(* CODESYS project SPT_Vision.library
   Company: Beckhoff Automation LLC
   DefaultNamespace: SPT_Vision
   Version: 3.0.0
   Placeholder: SPT Vision
   Title: SPT Vision

Project tree, tasks and I/O mapping:
  libraries: SPT Base Types, * (Beckhoff Automation LLC); Tc2_Standard, * (Beckhoff Automation GmbH); Tc2_System, * (Beckhoff Automation GmbH); Tc3_Module, * (Beckhoff Automation GmbH); Tc3_Vision, * (Beckhoff Automation GmbH); SPT Event Logger, * (Beckhoff Automation LLC); Tc3_EventLogger, * (Beckhoff Automation GmbH); Tc2_Utilities, * (Beckhoff Automation GmbH); Tc2_EtherCAT, * (Beckhoff Automation GmbH)
  DUTs/
  GVLs/
  POUs/
    program MAIN [ST]
  Project Information/
    function F_GetCompany [ST]
    function F_GetTitle [ST]
    function F_GetVersion [ST]
  Version/
    global variables Global_Version
  Vision/
    DUTs/
      data type E_VisionTools
      data type ST_BlobResults
      data type ST_CameraReadWrite
      data type ST_Image2Video
      data type ST_VisionResults
    GVLs/
      global variables GVL_CameraDefinitions
      global variables GVL_Image2Video
      global variables GVL_VisionColor
    HMI/
      data type ST_VisionBase_Command
      data type ST_VisionBase_Config
      data type ST_VisionBase_HMI
      data type ST_VisionBase_Status
    PLC Task/
      function block FB_PlcCameraBase [ST]: CreateEvents, CyclicLogic, GetResults, Reset, RunVision, TriggerImage
    VisionTask/
      function block FB_CameraParameterBuffer [ST]: AddData, BufferCount, GetData, ReadData, ResetData
      function block FB_VideoPlaybackControl [ST]: Busy, Error, ErrorID, CyclicLogic, InitComplete, Execute, OnAlarmRaised, SubscribedEvents, SubscribeEvents, UnsubscribeEvents, AddImage, AlarmDelayTime, CameraID, FramesPerSecond, ImageReductionFactor, ImageSourceDirectory, VideoOutputDirectory, WriteImage
      function block FB_VisionCameraBase [ST]: LightBackground, ExposureAddress, GainAddress, CyclicLogic, HMICommunication, ProcessImage, ReadParamUDINT, SetParamUDINT
      function block FB_VisionCameraDetection [ST]: ProcessImage, Initialize
      function block FB_VisionCameraMonitor [ST]: CameraID, FramesPerSecond, ImageSourceDirectory, VideoOutputDirectory, CyclicLogic, Initialize, ProcessImage
      interface I_CameraBase: CyclicLogic, ProcessImage
    global variables Parameters_Vision
  VISUs/
*)

// Vision/DUTs/E_VisionTools
{attribute 'qualified_only'}
{attribute 'strict'}
TYPE E_VisionTools :
(
	Blob,
	Contour,
	Color
);
END_TYPE

// Vision/DUTs/ST_BlobResults
TYPE ST_BlobResults :
	STRUCT
		Area		   : LREAL;
		CenterOfMass   : TcVnPoint2_LREAL;
		Circularity	   : LREAL;
		Convexity	   : LREAL;
		Eccentricity   : LREAL;
		ExtremePoint   : TcVnPoint2_LREAL;
		InertiaRatio   : LREAL;
		Moments		   : TcVnMoments;
		Orientation	   : TcVnRotatedRectangle;
		OrientationExp : TcVnRotatedRectangle;
		Perimeter	   : LREAL;
		Roundness	   : LREAL;
	END_STRUCT
END_TYPE

// Vision/DUTs/ST_CameraReadWrite
TYPE ST_CameraReadWrite :
	(*CameraCommand consists of Camera parameter address in HEX(byte)
	AND the data TO be written TO that address in decimal (UDINT).*)
	STRUCT
		CamAddress : UDINT;
		CamData	   : UDINT;
		Valid	   : BOOL;
	END_STRUCT
END_TYPE

// Vision/DUTs/ST_Image2Video
TYPE ST_Image2Video :
	STRUCT
		VideoPathSource : STRING;
		ImagePathSource : STRING;
		VideoFilename	: STRING;
		VideoCreate		: BOOL;
		VideoCreated	: BOOL;
		VideoFPS		: UINT;
		Heartbeat		: BOOL;
	END_STRUCT
END_TYPE

// Vision/DUTs/ST_VisionResults
{attribute 'pack_mode' := '1'}
TYPE ST_VisionResults :
	STRUCT
		x		 : LREAL; //x offset in image
		y		 : LREAL; //y offset in image
		c		 : LREAL; //Rotation about Z
		Pass	 : BOOL;  //Pass/Fail bit
		Distance : LREAL; //Distance in measurement
	END_STRUCT
END_TYPE

// Vision/HMI/ST_VisionBase_Command
TYPE ST_VisionBase_Command :
	STRUCT
		StartAquisition : BOOL;
		StopAquisition	: BOOL;
		Trigger			: BOOL;
	END_STRUCT
END_TYPE

// Vision/HMI/ST_VisionBase_Config
TYPE ST_VisionBase_Config :
	STRUCT
		Gain			  : UDINT;
		SetGain			  : BOOL;
		ReadGain		  : BOOL;
		ReadGainValue	  : UDINT;
		Exposure		  : UDINT;
		SetExposure		  : BOOL;
		ReadExposure	  : BOOL;
		ReadExposureValue : UDINT;
	END_STRUCT
END_TYPE

// Vision/HMI/ST_VisionBase_HMI
TYPE ST_VisionBase_HMI :
	STRUCT
		Config	: ST_VisionBase_Config;
		Command : ST_VisionBase_Command;
		Status	: ST_VisionBase_Status;
	END_STRUCT
END_TYPE

// Vision/HMI/ST_VisionBase_Status
 
TYPE ST_VisionBase_Status :
	STRUCT
		VisionRunning : BOOL;
		CameraState	  : ETcVnCameraState;
		ElementsFound : UDINT;
	END_STRUCT
END_TYPE

// Version/Global_Version
{attribute 'TcGenerated'}
{attribute 'no-analysis'}
{attribute 'linkalways'}
// This function has been automatically generated from the project information.
VAR_GLOBAL CONSTANT
	{attribute 'const_non_replaced'}
	stLibVersion_SPT_Vision : ST_LibVersion := (iMajor := 3, iMinor := 0, iBuild := 0, iRevision := 0, nFlags := 0, sVersion := '3.0.0');
END_VAR

// Vision/GVLs/GVL_CameraDefinitions
{attribute 'qualified_only'}
VAR_GLOBAL CONSTANT
	
	// Baseler ACE camera 
	// Analog Controls - Gain
	M180_GAIN_ADDRESS	   : UDINT := 16#00020024; // only writeable if Gain Auto is off (220-850)

	// Acquisition - Trigger
	M180_TRIGGER_MODE_ADDRESS	: UDINT := 16#00040204; // 0= Off 1 = On
	M180_TRIGGER_SOURCE_ADDRESS : UDINT := 16#00040244; // 0 = software 1 = line(hardware)

	// Acquisition - Exposure
	M180_EXPOSURE_TIME_ADDRESS : UDINT := 16#00040464; // 24-1000000us 

	// AOI Controls
	M180_WIDTH_ADDRESS	  : UDINT := 16#00030204; // 1 - Camera width based on Binning
	M180_HEIGHT_ADDRESS	  : UDINT := 16#00030224; // 1 - Camera height based on Binning
	M180_X_OFFSET_ADDRESS : UDINT := 16#00030244; // pixel offset to be used if the width is smaller than max-adjust view
	M180_Y_OFFSET_ADDRESS : UDINT := 16#00030264; // pixel offset to be used if the height is smaller than max-adjust view
END_VAR

// Vision/GVLs/GVL_Image2Video
{attribute 'qualified_only'}
VAR_GLOBAL
	NumberOfCameras	   : UINT := Parameters_Vision.MAX_NUMBER_CAMERAS;
	CameraData		   : ARRAY[1..Parameters_Vision.MAX_NUMBER_CAMERAS] OF ST_Image2Video;
END_VAR

// Vision/GVLs/GVL_VisionColor
{attribute 'qualified_only'}
{attribute 'strict'}
VAR_GLOBAL
	ColorWhite	 : TcVnVector4_LREAL := [255, 255, 255, 255];
	ColorBlack	 : TcVnVector4_LREAL := [0, 0, 0, 255];
	ColorGreen	 : TcVnVector4_LREAL := [0, 175, 0, 255];
	ColorBlue	 : TcVnVector4_LREAL := [0, 0, 255, 255];
	ColorRed	 : TcVnVector4_LREAL := [255, 0, 0, 255];
	ColorMagenta : TcVnVector4_LREAL := [255, 0, 255, 255];
END_VAR

// Vision/Parameters_Vision
{attribute 'qualified_only'}
VAR_GLOBAL CONSTANT
	MAX_RESULTS_BUFFER_BYTES   : UDINT := 1000;
	MAX_NUMBER_CAMERAS : USINT := 1;
	MAX_NUMBER_IMAGES_2_VIDEO : UINT := 200;
END_VAR

// POUs/MAIN
PROGRAM MAIN
VAR
END_VAR

END_PROGRAM

// Project Information/F_GetCompany
// This function has been automatically generated from the project information.
{attribute 'signature_flag' := '1073741824'}
{attribute 'TcGenerated'}
{attribute 'no-analysis'}
FUNCTION F_GetCompany : WSTRING
VAR_INPUT
	
END_VAR

F_GetCompany := "Beckhoff Automation LLC";

END_FUNCTION

// Project Information/F_GetTitle
// This function has been automatically generated from the project information.
{attribute 'signature_flag' := '1073741824'}
{attribute 'TcGenerated'}
{attribute 'no-analysis'}
FUNCTION F_GetTitle : WSTRING
VAR_INPUT
	
END_VAR

F_GetTitle := "SPT Vision";

END_FUNCTION

// Project Information/F_GetVersion
// This function has been automatically generated from the project information.
{attribute 'signature_flag' := '1073741824'}
{attribute 'TcGenerated'}
{attribute 'no-analysis'}
FUNCTION F_GetVersion : ST_LibVersion
VAR_INPUT
	
END_VAR

F_GetVersion.iMajor := 3;
F_GetVersion.iMinor := 0;
F_GetVersion.iBuild := 0;
F_GetVersion.iRevision := 0;
F_GetVersion.sVersion := '3.0.0';
F_GetVersion.nFlags := 0;

END_FUNCTION

// Vision/PLC Task/FB_PlcCameraBase
FUNCTION_BLOCK FB_PlcCameraBase EXTENDS FB_ComponentBase
VAR
	//Outputs
	SoftwareTrigger	   AT %Q* : BOOL;
	_RunVision		   AT %Q* : BOOL;
	_Reset			   AT %Q* : BOOL;

	//Inputs
	CameraState			 AT %I* : ETcVnCameraState;
	ResultsAvailable	 AT %I* : BOOL;
	NumberOfResults		 AT %I* : UDINT;
	Results				 AT %I* : ARRAY[1..Parameters_Vision.MAX_RESULTS_BUFFER_BYTES] OF BYTE;
	VisionError			 AT %I* : BOOL;
	VisionErrorID		 AT %I* : UDINT;

	
	VisionAlarms : ARRAY[1..5] OF FB_TcAlarm;
END_VAR

//! @summary Initializes event function blocks using this components's name
METHOD PROTECTED CreateEvents

//! @description This method is called by <c>Initialize()</c> as required
SUPER^.CreateEvents();

F_CreateAllEventsInClass(Alarms		:= VisionAlarms,
						 ClassSize	:= SIZEOF(TC_EVENTS.VisionBaseAlarms),
						 pInitEvent := ADR(TC_EVENTS.VisionBaseAlarms.InitReferenceEvent),
						 Prefix		:= Name);
END_METHOD

//! @summary This method serves as the entry point for all underlying FB logic
METHOD PUBLIC CyclicLogic

//! @description This method should be called cyclically by descendant function blocks by invoking <c>SUPER^.CyclicLogic()</c>.  Alternatively, the contents of this method could be reimplemented entirely in which case a call to this method would not be necessary.
SUPER^.CyclicLogic();

// Monitor camera error here
IF VisionError AND NOT VisionAlarms[E_VisionBaseAlarms.CameraFault].bRaised THEN
	VisionAlarms[E_VisionBaseAlarms.CameraFault].Raise(0);
ELSIF NOT VisionError AND VisionAlarms[E_VisionBaseAlarms.CameraFault].bRaised THEN
	VisionAlarms[E_VisionBaseAlarms.CameraFault].Clear(0, 0);
END_IF

_Error := VisionAlarms[E_VisionBaseAlarms.CameraFault].bRaised;
IF _Error THEN
	_ErrorID := VisionErrorID;
//ELSE
//	_ErrorID := 0;
END_IF

_Busy := _RunVision;
END_METHOD

METHOD GetResults : BOOL
VAR_IN_OUT
	ResultArray : ARRAY[1..Parameters_Vision.MAX_RESULTS_BUFFER_BYTES] OF BYTE;
	Number		: UDINT;
END_VAR

VAR_INST
	ResultsAvailable_RTRIG : R_TRIG;
END_VAR
GetResults := FALSE;
ResultsAvailable_RTRIG(CLK := ResultsAvailable);
IF ResultsAvailable_RTRIG.Q THEN
	IF SIZEOF(ResultArray) < SIZEOF(Results) THEN
		MEMCPY(ADR(ResultArray), ADR(Results), SIZEOF(ResultArray));
	ELSE
		MEMCPY(ADR(ResultArray), ADR(Results), SIZEOF(Results));
	END_IF

	IF NumberOfResults * SIZEOF(Results) > SIZEOF(ResultArray) THEN
		; ///Handle alarm
	END_IF

	Number	   := NumberOfResults;
	GetResults := TRUE;
END_IF
END_METHOD

//! @summary Clears error flags and error IDs for this component
METHOD PUBLIC Reset : BOOL
//Return the value from the base FB Reset()
Reset := SUPER^.Reset();

// Clear the Vision Alarms
F_ClearAllEventsInClass(Alarms:=VisionAlarms);

// Set the Error ID to 0
_ErrorID := 0;
END_METHOD

PROPERTY RunVision : BOOL
SET
_RunVision := RunVision;
SoftwareTrigger := false;
END_SET
END_PROPERTY

PROPERTY TriggerImage : BOOL
SET
SoftwareTrigger := TriggerImage;
END_SET
END_PROPERTY

END_FUNCTION_BLOCK

// Vision/VisionTask/FB_CameraParameterBuffer
FUNCTION_BLOCK FB_CameraParameterBuffer
VAR
	buffer : FB_MemRingBuffer;
	bufferData : ARRAY[0..100] OF UDINT;
END_VAR

METHOD AddData : BOOL
VAR_INPUT
	data : ST_CameraReadWrite;
END_VAR
buffer(pWrite:=ADR(data),cbWrite:=SIZEOF(data));

buffer.A_AddTail();
END_METHOD

PROPERTY BufferCount : UDINT
GET
BufferCount := buffer.nCount;
END_GET
END_PROPERTY

METHOD GetData
VAR_OUTPUT
	data : ST_CameraReadWrite;
END_VAR
buffer(pRead := ADR(data), cbRead := SIZEOF(data));
buffer.A_GetHead();
END_METHOD

METHOD ReadData : BOOL
VAR_OUTPUT
	data : ST_CameraReadWrite;
END_VAR
buffer(pRead := ADR(data), cbRead := SIZEOF(data));
buffer.A_GetHead();
buffer.A_RemoveHead();
END_METHOD

METHOD ResetData : BOOL
VAR_INPUT
END_VAR
buffer(pBuffer:=ADR(bufferData),cbBuffer:=SIZEOF(bufferData));
buffer.A_Reset();
END_METHOD

END_FUNCTION_BLOCK

// Vision/VisionTask/FB_VideoPlaybackControl
FUNCTION_BLOCK FB_VideoPlaybackControl EXTENDS FB_ListenerBase2 IMPLEMENTS I_CyclicFB
VAR
	//Base FB
	_Busy	 : BOOL := TRUE;
	_Error	 : BOOL;
	_ErrorID : UDINT;

	//Cyclic FB
	_InitComplete : BOOL;

	// Video Playback Control
	_CameraID : UINT;

	//EnableImagesToBuffer : BOOL;
	TriggerVideoCapture : BOOL;
	VideoCaptureState	: INT;

	// Ring Buffer information
	BufferImageRing : ARRAY[1..Parameters_Vision.MAX_NUMBER_IMAGES_2_VIDEO] OF ITcVnImage;
	BufferIndex		: INT := 1;

	//BufferImageSaveIndex	  : UINT;
	WriteImageWaitResult	  : BOOL;
	ipImageForVideoRingBuffer : ITcVnImage;
	ipImageToSave			  : ITcVnImage;
	WriteFileState			  : INT;
	sImageToSaveName		  : STRING;
	fbWriteImage			  : FB_VN_WriteImage;
	SysTimeAtFileWrite		  : ULINT;
	_fbEvent				  : FB_TcEvent;
	sFileName1				  : T_MaxString;

	//Properties
	_ImageReductionFactor : LREAL := 1; // This is the amount of reduction to image for making video Default := 1;
	_ImageSourceDirectory : STRING;
	_VideoOutputDirectory : STRING;
	_FramesPerSecond	  : UINT;

	//Alarm data
	sJsonAttribute	 : STRING(10000);
	JSONFilter		 : FB_TcEventFilter;
	JSONString		 : T_MaxString := '{"CreateVideo": 1}';
	_Subscribe		 : BOOL		   := TRUE;
	_Unsubscribe	 : BOOL;
	_Subscribed		 : BOOL;
	MissedEventCount : UDINT;

	//Image count value
	ImageWriteCount : UINT;

	//Delay after alarm to wait then do work
	AlarmDelay		: TON;
	_AlarmDelayTime : TIME;
	StopImageAdding : BOOL;
END_VAR

PROPERTY Busy : BOOL
GET
Busy := _Busy;
END_GET
END_PROPERTY

PROPERTY Error : BOOL
GET
Error := _Error;
END_GET
END_PROPERTY

PROPERTY ErrorID : UDINT
GET
ErrorID := _ErrorID;
END_GET
END_PROPERTY

METHOD CyclicLogic
VAR
	hr				: HRESULT;
	tmpIndex		: INT;
	systemTimeNow	: TIMESTRUCT;
	tmpString		: STRING;
	EventTimestamp1 : TimeStruct;
	sDump			: STRING;
END_VAR

VAR_INST
	x : INT;
END_VAR
IF NOT _InitComplete THEN
	_InitComplete := TRUE;
END_IF

// Call the Listener Execute
Execute();
IF _Subscribe THEN
	_Subscribe := FALSE;
	JSONFilter.Clear().JsonAttribute.Value.EqualTo(JSONString); //define all events (messages and alarms) from this eventclass   
	hr := Subscribe2(JSONFilter);								//subscribe to retrieve defined events
	IF SUCCEEDED(hr) THEN
		_Subscribed := TRUE;
	END_IF
END_IF

IF _Unsubscribe THEN
	_Unsubscribe := FALSE;
	hr			 := Unsubscribe();
	IF SUCCEEDED(hr) THEN
		_Subscribed := FALSE;
	END_IF
END_IF

CASE VideoCaptureState OF
	0:
		IF TriggerVideoCapture THEN
			x				  := 1;
			VideoCaptureState := 10;
		END_IF

	10:
		IF AlarmDelay.Q THEN
			StopImageAdding := TRUE;
			VideoCaptureState := 15;
		END_IF
	
	15:	
		tmpIndex := BufferIndex + x - 1;
		IF tmpIndex > TO_INT(Parameters_Vision.MAX_NUMBER_IMAGES_2_VIDEO) THEN
			tmpIndex := tmpIndex - TO_INT(Parameters_Vision.MAX_NUMBER_IMAGES_2_VIDEO);
		END_IF

		IF WriteImage(Index := x, BufferImageSaveNameIndex := TmpIndex) THEN
			x := x + 1;
		END_IF

		IF x > TO_INT(Parameters_Vision.MAX_NUMBER_IMAGES_2_VIDEO) THEN
			TriggerVideoCapture := FALSE;
			StopImageAdding := FALSE;
			VideoCaptureState	:= 20;
		END_IF

	20:
		EventTimestamp1 := FILETIME64_TO_SYSTEMTIME(_fbevent.nTimestamp);
		sFileName1		:= SYSTEMTIME_TO_STRING(EventTimestamp1);
		FindAndReplaceChar(ADR(sFileName1),
						   ':',
						   '-',
						   ADR(sFileName1),
						   SIZEOF(sFileName1));

		FindAndSplitChar(sSeparatorChar	  := '.',
						 pSrcString		  := ADR(sFileName1),
						 pLeftString	  := ADR(sFileName1),
						 nLeftSize		  := SIZEOF(sFileName1),
						 pRightString	  := ADR(sDump),
						 nRightSize		  := SIZEOF(sDump),
						 bSearchFromRight := FALSE);

		sFileName1											:= CONCAT(sFileName1, '.avi');
		GVL_Image2Video.CameraData[_CameraID].VideoFilename := sFileName1;
		GVL_Image2Video.CameraData[_CameraID].VideoCreate	:= TRUE;
		VideoCaptureState									:= 30;

	30:
		IF GVL_Image2Video.CameraData[_CameraID].VideoCreated THEN
			GVL_Image2Video.CameraData[_CameraID].VideoCreate  := FALSE;
			GVL_Image2Video.CameraData[_CameraID].VideoCreated := FALSE;
			VideoCaptureState								   := 0;
		END_IF
END_CASE

IF GVL_Image2Video.CameraData[_CameraID].Heartbeat THEN
	GVL_Image2Video.CameraData[_CameraID].Heartbeat := FALSE;
END_IF

AlarmDelay(IN:= VideoCaptureState =10, PT:=_AlarmDelayTime);

GVL_Image2Video.CameraData[_CameraID].VideoPathSource := _VideoOutputDirectory;
GVL_Image2Video.CameraData[_CameraID].ImagePathSource := _ImageSourceDirectory;
GVL_Image2Video.CameraData[_CameraID].VideoFPS		  := _FramesPerSecond;
END_METHOD

PROPERTY InitComplete : BOOL
GET
InitComplete := _InitComplete;
END_GET
END_PROPERTY

METHOD Execute : HRESULT
VAR_INPUT
END_VAR
Execute := SUPER^.Execute();
END_METHOD

METHOD OnAlarmRaised : HRESULT
VAR_INPUT
	fbEvent : REFERENCE TO FB_TcEvent;
END_VAR

VAR 
	hr : HRESULT;
END_VAR
// This is where we actually do the work
IF NOT TriggerVideoCapture THEN
	TriggerVideoCapture := TRUE;
	ImageWriteCount := 1;
	hr					:= fbEvent.GetJsonAttribute(sJsonAttribute, SIZEOF(sJsonAttribute));
	_fbEvent:=fbevent;
ELSE
	MissedEventCount := MissedEventCount + 1;
END_IF

OnAlarmRaised := S_OK;
END_METHOD

PROPERTY SubscribedEvents : BOOL
GET
SubscribedEvents := _Subscribed;
END_GET
END_PROPERTY

PROPERTY SubscribeEvents : BOOL
SET
_Subscribe := SubscribeEvents;
END_SET
END_PROPERTY

PROPERTY UnsubscribeEvents : BOOL
SET
_Unsubscribe := UnsubscribeEvents;
END_SET
END_PROPERTY

METHOD AddImage : BOOL
VAR_INPUT
	ipImageIn : ITcVnImage; // Image to be added to buffer
END_VAR

VAR
	hr						  : HRESULT;
	hrWD1					  : HRESULT;
	tStop1					  : DINT := 20000;
	tRest1					  : DINT;
	ImageInfo				  : TcVnImageInfo;
	ImagePixelFormatChannels  : BYTE;
	ImageEffectivePixelSize	  : UINT;
	ImageInWidth			  : UDINT;
	ImageInHeight			  : UDINT;
	ImageSmallWidth			  : UDINT;
	ImageSmallHeight		  : UDINT;
END_VAR
IF NOT StopImageAdding THEN
	hr						 := F_VN_GetImageInfo(ipImage := ipImageIn, stImageInfo := ImageInfo, hrPrev := S_OK);
	ImagePixelFormatChannels := ImageInfo.stPixelFormat.nChannels;
	ImageEffectivePixelSize	 := ImageInfo.stPixelFormat.nElementSize;
	ImageInWidth			 := ImageInfo.nWidth;
	ImageInHeight			 := ImageInfo.nHeight;
	IF _ImageReductionFactor <> 1 THEN
		ImageSmallWidth	 := LREAL_TO_UDINT(UDINT_TO_LREAL(ImageInWidth) * _ImageReductionFactor);
		ImageSmallHeight := LREAL_TO_UDINT(UDINT_TO_LREAL(ImageInHeight) * _ImageReductionFactor);

		// Image Width and Height must be even for video conversion
		IF (ImageSmallWidth MOD 2) <> 0 THEN // Check if "Odd"
			ImageSmallWidth := ImageSmallWidth - 1;
		END_IF

		IF (ImageSmallHeight MOD 2) <> 0 THEN // Check if "Odd"
			ImageSmallHeight := ImageSmallHeight - 1;
		END_IF

		hr := F_VN_ResizeImage(ipImageIn,
							   ipImageForVideoRingBuffer,
							   ImageSmallWidth,
							   ImageSmallHeight,
							   1,
							   hr);
	ELSE
		hr := F_VN_CopyImage(ipImageIn, ipImageForVideoRingBuffer, hr);
	END_IF

	// Check to see if images are in memory
	//hr := FW_SafeRelease(ADR(BufferImageRing[BufferIndex]));
	//IF BufferImageRing[BufferIndex] <> 0 THEN
	//	FW_SafeRelease(ADR(BufferImageRing[BufferIndex]));
	//END_IF
	
	
	hrWD1		:= F_VN_StartRelWatchdog(tStop1, S_OK);
	hr			:= F_VN_CopyImage(ipImageForVideoRingBuffer, BufferImageRing[BufferIndex], S_OK);
	hrWD1		:= F_VN_StopWatchdog(hrWD1, tRest => tRest1);
	BufferIndex := BufferIndex + 1;
	IF BufferIndex > Parameters_Vision.MAX_NUMBER_IMAGES_2_VIDEO THEN
		BufferIndex := 1;
	END_IF
END_IF
END_METHOD

PROPERTY AlarmDelayTime : TIME
SET
_AlarmDelayTime := AlarmDelayTime;
END_SET
END_PROPERTY

PROPERTY CameraID : UINT
SET
_CameraID := CameraID;
END_SET
END_PROPERTY

PROPERTY FramesPerSecond : UINT
SET
_FramesPerSecond := FramesPerSecond;
END_SET
END_PROPERTY

PROPERTY ImageReductionFactor : LREAL
SET
_ImageReductionFactor := ImageReductionFactor;
END_SET
END_PROPERTY

PROPERTY ImageSourceDirectory : STRING
SET
_ImageSourceDirectory := ImageSourceDirectory;
END_SET
END_PROPERTY

PROPERTY VideoOutputDirectory : STRING
SET
_VideoOutputDirectory := VideoOutputDirectory;
END_SET
END_PROPERTY

METHOD WriteImage : BOOL
VAR_INPUT
	BufferImageSaveNameIndex : INT;
	Index					 : INT;
END_VAR

VAR
	SysTimeAtImageSave : ULINT;
END_VAR
CASE WriteFileState OF
	0:
		sImageToSaveName := CONCAT(STR1 := _ImageSourceDirectory, '\Image');
		CASE Index OF // Add leading zeros to index number of image name
			0..9:
				sImageToSaveName := CONCAT(sImageToSaveName, '000');
				sImageToSaveName := CONCAT(sImageToSaveName, ULINT_TO_STRING(Index));

			10..99:
				sImageToSaveName := CONCAT(sImageToSaveName, '00');
				sImageToSaveName := CONCAT(sImageToSaveName, ULINT_TO_STRING(Index));

			100..999:
				sImageToSaveName := CONCAT(sImageToSaveName, '0');
				sImageToSaveName := CONCAT(sImageToSaveName, ULINT_TO_STRING(Index));

		ELSE
			sImageToSaveName := CONCAT(sImageToSaveName, ULINT_TO_STRING(Index));
		END_CASE;

		sImageToSaveName	:= CONCAT(sImageToSaveName, '.png');
		ipImageToSave		:= BufferImageRing[BufferImageSaveNameIndex];
		SysTimeAtImageSave	:= F_GetSystemTime();
		WriteFileState		:= 10;

	10:
		// sFilePath must contain the full path, image name and type
		fbWriteImage(ipImage := ipImageToSave, sFilePath := sImageToSaveName, nTimeout := T#500MS,bWrite := TRUE);
		IF NOT fbWriteImage.bBusy THEN
			fbWriteImage(sFilePath := sImageToSaveName, bWrite := FALSE);
			WriteFileState := 0;
			WriteImage := TRUE;
		END_IF

ELSE
	WriteFileState := 0;
END_CASE

(*//bSaveImageNow := FALSE;
WriteImageWaitResult := TRUE;

// sFilePath must contain the full path, image name and type
fbWriteImage(ipImage   := ipImageToSave,
			 sFilePath := sImageToSaveName,
			 bWrite	   := TRUE,
			 nTimeout  := T#500MS);

IF NOT fbWriteImage.bBusy AND NOT fbWriteImage.bError THEN
	fbWriteImage(bWrite := FALSE, sFilePath := sImageToSaveName);
	WriteImage := TRUE;
END_IF*)
END_METHOD

END_FUNCTION_BLOCK

// Vision/VisionTask/FB_VisionCameraBase
FUNCTION_BLOCK ABSTRACT FB_VisionCameraBase EXTENDS FB_ComponentBase IMPLEMENTS I_CameraBase
VAR
	// Vision Related
	hr		   : HRESULT;
	Camera	   : FB_VN_SimpleCameraControl;
	ipImageIn  : ITcVnImage;
	ImageCount : ULINT;

	//Inputs to Camera
	RunVision		AT %I* : BOOL;
	SoftwareTrigger AT %I* : BOOL;
	Reset			AT %I* : BOOL;

	//Outputs From Camera (Property)
	CameraState		 AT %Q* : ETcVnCameraState;
	ResultsAvailable AT %Q* : BOOL;
	NumberOfResults	 AT %Q* : UDINT;
	Results			 AT %Q* : ARRAY[1..Parameters_Vision.MAX_RESULTS_BUFFER_BYTES] OF BYTE;
	VisionError		 AT %Q* : BOOL;
	VisionErrorID	 AT %Q* : UDINT;

	//Read Write Data
	_ReadData		: BOOL;
	_ReadAddress	: UDINT;
	_WriteData		: BOOL;
	_WriteValue		: UDINT;
	_WriteAddress	: UDINT;
	_ReadDataResult : BOOL;
	_ReadDataValue	: UDINT;
	_ReadDataValid	: BOOL;
	_WriteDataDone	: BOOL;

	//Camera Addresses
	_ExposureAddress : UDINT; //Default is zero and checked when asked to write
	_GainAddress	 : UDINT;

	//Camera Parameter Read/Write Section ******************************************************************
	WriteCamera			  : FB_VN_WriteRegister_UDINT;
	ReadCamera			  : FB_VN_ReadRegister_UDINT;
	ReadValue			  : UDINT;
	ReadCamera_FTRIG	  : F_TRIG;
	ReadCameraError_RTRIG : R_TRIG;

	// Timing Statistics
	SysTimeAtImageArrive : ULINT; // system time units = 1 nS
	SysTimeAtTrigger	 : ULINT; // system time units = 1 nS
	SysTimeAfterProcess	 : ULINT; // system time units = 1 nS
	_ProcessTime		 : LREAL;
	_TriggerToImageTime	 : LREAL;
	_TotalTime			 : LREAL;

	//Read/Write params
	tmpCamParamRead		  : ST_CameraReadWrite;
	tmpCamReadData		  : ST_CameraReadWrite;
	ReadCameraData_RTRIG  : R_TRIG;
	WriteCameraData_RTRIG : R_TRIG;

	//Trigger support
	SoftwareTrigger_RTRIG : R_TRIG;
	HMI_Trigger			  : BOOL;

	//HMI
	VisionBase_HMI : ST_VisionBase_HMI;

	//Generic Results
	FeedbackResults : ARRAY[1..100] OF ST_VisionResults;

	// Image Infos
	PixelFormat : TcVnPixelFormat;

	//HRESULT
	hrFunc : HRESULT;

	// Image Interfaces	
	ipImageInDisp		 : ITcVnDisplayableImage;
	ipImageRes			 : ITcVnImage;
	ipImageResDisp		 : ITcVnDisplayableImage;
	ipImageWork			 : ITcVnImage;
	ipImageThresholdDisp : ITcVnDisplayableImage;

	//Properties
	_LightBackground : BOOL;

	// Parameters for Blob
	BlobParameters : TcVnParamsBlobDetection;

	// Watchdog
	hrWD	  : HRESULT;
	tStop	  : DINT := 5000;
	tRest	  : DINT;
	nFraction : UDINT;

	// Sample Specific Variables
	ipContourList : ITcVnContainer;
END_VAR

PROPERTY LightBackground : BOOL
GET
LightBackground := _LightBackground;
END_GET
SET
_LightBackground := LightBackground;
END_SET
END_PROPERTY

PROPERTY ExposureAddress : UDINT
SET
_ExposureAddress := ExposureAddress;
END_SET
END_PROPERTY

PROPERTY GainAddress : UDINT
SET
_GainAddress := GainAddress;
END_SET
END_PROPERTY

METHOD PUBLIC CyclicLogic
SUPER^.CyclicLogic();

// Do the camera logic
CameraState := Camera.GetState();
CASE CameraState OF
	// Initializing States to get to opened
	TCVN_CS_INITIAL, TCVN_CS_INITIALIZING, TCVN_CS_INITIALIZED, TCVN_CS_OPENING:
		hr := Camera.StartAcquisition();
		IF CameraState = TCVN_CS_INITIALIZED THEN
			VisionError := FALSE;
		END_IF

	// In opened, continue if application asks to run
	TCVN_CS_OPENED:
		IF RunVision THEN
			hr := Camera.StartAcquisition();
		END_IF

	// Always call another StartAquisition when in that state
	TCVN_CS_STARTACQUISITION:
		hr := Camera.StartAcquisition();

	// Response to the Triggering is to TriggerImage again
	TCVN_CS_TRIGGERING:
		hr := Camera.TriggerImage();

	// Waiting for image or application asked to stop running
	TCVN_CS_ACQUIRING:
		hr := Camera.GetCurrentImage(ipImageIn);

		// Check if new Image was received
		IF SUCCEEDED(hr) AND ipImageIn <> 0 THEN
			SysTimeAtImageArrive := F_GetActualDcTime64(); // get system time at new image
			ImageCount			 := ImageCount + 1;
			ProcessImage();
			SysTimeAfterProcess := F_GetActualDcTime64();
			ResultsAvailable	:= TRUE;
			_ProcessTime		:= TO_LREAL(SysTimeAfterProcess - SysTimeAtImageArrive) / TO_LREAL(Tc2_EtherCAT.EC_DCTIME_TICKSPERMSEC64);
			_TriggerToImageTime := TO_LREAL(SysTimeAtImageArrive - SysTimeAtTrigger) / TO_LREAL(Tc2_EtherCAT.EC_DCTIME_TICKSPERMSEC64);
			_TotalTime			:= TO_LREAL(SysTimeAfterProcess - SysTimeAtTrigger) / TO_LREAL(Tc2_EtherCAT.EC_DCTIME_TICKSPERMSEC64);
		ELSIF NOT RunVision THEN
			Camera.StopAcquisition();
		END_IF

	// Stop acqusition requires another call to StopAcquisiton
	TCVN_CS_STOPACQUISITION:
		hr := Camera.StopAcquisition();

	///UH oh.  We are in an error state  try to reset and initialize
	TCVN_CS_ERROR:
		VisionError			:= TRUE;
		hr := Camera.Reset();
END_CASE

//Handle Triggering here
SoftwareTrigger_RTRIG(CLK := (SoftwareTrigger OR HMI_Trigger));
IF SoftwareTrigger_RTRIG.Q THEN
	ResultsAvailable := FALSE;
	hr				 := Camera.TriggerImage();
	IF SUCCEEDED(hr) THEN
		SysTimeAtTrigger := F_GetActualDcTime64();
	END_IF
END_IF

(* Read/Write Camera Data ****************************************************************************
 Check for data in Process Image*)
ReadCameraData_RTRIG(CLK := _ReadData);
IF ReadCameraData_RTRIG.Q THEN
	_ReadDataResult		:= FALSE;
	ReadCamera.nAddress := _ReadAddress;
	ReadCamera.bRead	:= TRUE;
END_IF

ReadCamera(nEndian := 0, nTimeout := T#5S);
ReadCameraError_RTRIG(Clk := ReadCamera.bError AND ReadCamera.bRead AND NOT ReadCamera.bBusy);
ReadCamera.bRead := FALSE;
ReadCamera_FTRIG(CLK := ReadCamera.bBusy);
IF ReadCamera_FTRIG.Q OR ReadCameraError_RTRIG.Q THEN
	IF ReadCamera.bError THEN //ADSERR_DEVICE_BUSY
		_ReadDataResult := TRUE;
		_ReadDataValid	:= FALSE;
	ELSE
		_ReadDataResult := TRUE;
		_ReadDataValue	:= ReadCamera.nValue;
		_ReadDataValid	:= TRUE;
	END_IF
END_IF

WriteCameraData_RTRIG(CLK := _WriteData);

// Check Queue of parameters and Write to Camera
IF WriteCameraData_RTRIG.Q THEN
	_WriteDataDone		 := FALSE;
	WriteCamera.nAddress := _WriteAddress;
	WriteCamera.nValue	 := _WriteValue;
	WriteCamera.bWrite	 := TRUE;
END_IF

WriteCamera(nEndian := 0, nTimeout := T#5S);
WriteCamera.bWrite := FALSE;
IF _WriteData AND (NOT WriteCamera.bBusy OR WriteCamera.bError) THEN
	_WriteDataDone := TRUE;
END_IF

HMICommunication();
END_METHOD

METHOD PROTECTED HMICommunication
VAR_INPUT
END_VAR

VAR_INST
	Trigger_RTRIG	   : R_TRIG;
	ReadExposure_RTRIG : R_TRIG;
	ReadGain_RTRIG	   : R_TRIG;
	SetExposure_RTRIG  : R_TRIG;
	SetGain_RTRIG	   : R_TRIG;
	ReadGain		   : BOOL;
	ReadExposure	   : BOOL;
	SetGain			   : BOOL;
	SetExposure		   : BOOL;
END_VAR
Trigger_RTRIG(CLK := VisionBase_HMI.Command.Trigger);
ReadExposure_RTRIG(CLK := VisionBase_HMI.Config.ReadExposure);
ReadGain_RTRIG(CLK := VisionBase_HMI.Config.ReadGain);
SetExposure_RTRIG(CLK := VisionBase_HMI.Config.SetExposure);
SetGain_RTRIG(CLK := VisionBase_HMI.Config.SetGain);

// handle the request to run vision
IF ComponentBase_HMI.Status.HMIControlAvailable THEN
	IF VisionBase_HMI.Command.StartAquisition THEN
		RunVision := TRUE;
	ELSIF VisionBase_HMI.Command.StopAquisition THEN
		RunVision := FALSE;
	END_IF

	IF ReadExposure_RTRIG.Q AND NOT _ReadData THEN
		ReadExposure := TRUE;
		_ReadAddress := _ExposureAddress;
		_ReadData	 := TRUE;
	ELSIF _ReadDataResult AND ReadExposure THEN
		_ReadData								:= FALSE;
		_ReadDataResult							:= FALSE;
		ReadExposure							:= FALSE;
		VisionBase_HMI.Config.ReadExposureValue := _ReadDataValue;
	END_IF

	IF ReadGain_RTRIG.Q AND NOT _ReadData THEN
		ReadGain	 := TRUE;
		_ReadAddress := _GainAddress;
		_ReadData	 := TRUE;
	ELSIF _ReadDataResult AND ReadGain THEN
		_ReadData							:= FALSE;
		_ReadDataResult						:= FALSE;
		ReadGain							:= FALSE;
		VisionBase_HMI.Config.ReadGainValue := _ReadDataValue;
	END_IF

	IF SetExposure_RTRIG.Q AND NOT _WriteData THEN
		_WriteData	  := TRUE;
		SetExposure	  := TRUE;
		_WriteAddress := _ExposureAddress;
		_WriteValue	  := VisionBase_HMI.Config.Exposure;
	ELSIF _WriteDataDone AND SetExposure THEN
		SetExposure	   := FALSE;
		_WriteDataDone := FALSE;
		_WriteData	   := FALSE;
	END_IF

	IF SetGain_RTRIG.Q AND NOT _WriteData THEN
		SetGain		  := TRUE;
		_WriteData	  := TRUE;
		_WriteAddress := _GainAddress;
		_WriteValue	  := VisionBase_HMI.Config.Gain;
	ELSIF _WriteDataDone AND SetGain THEN
		SetGain		   := FALSE;
		_WriteDataDone := FALSE;
		_WriteData	   := FALSE;
	END_IF

	HMI_Trigger := Trigger_RTRIG.Q;
ELSE
	_ReadData		:= FALSE;
	_ReadDataResult := FALSE;
END_IF

VisionBase_HMI.Status.VisionRunning := RunVision;
VisionBase_HMI.Status.CameraState	:= CameraState;
VisionBase_HMI.Status.ElementsFound := NumberOfResults;
END_METHOD

METHOD PUBLIC  ProcessImage
// Convert Images into the necessary color space
hr := F_VN_GetPixelFormat(ipImageIn, PixelFormat, hr);
IF PixelFormat.nChannels = 3 THEN
	hr := F_VN_CopyImage(ipImageIn, ipImageRes, hr);
	hr := F_VN_ConvertColorSpace(ipImageRes,
								 ipImageIn,
								 TCVN_CST_RGB_TO_GRAY,
								 hr);
ELSE
	hr := F_VN_ConvertColorSpace(ipImageIn,
								 ipImageRes,
								 TCVN_CST_Gray_TO_RGB,
								 hr);
END_IF

// Image Segementation
IF _LightBackground THEN
	hr := F_VN_Threshold(ipImageIn,
						 ipImageWork,
						 BlobParameters.fMinThreshold,
						 255,
						 eThresholdType := TCVN_TT_BINARY_INV,
						 hr);
ELSE
	hr := F_VN_Threshold(ipImageIn,
						 ipImageWork,
						 BlobParameters.fMinThreshold,
						 255,
						 eThresholdType := TCVN_TT_BINARY,
						 hr);
END_IF

// Start Watchdog - DetectBlobs - Stop Watchdog
hrWD   := F_VN_StartRelWatchdog(tStop, S_OK);
hrFunc := F_VN_DetectBlobs(ipSrcImage	  := ipImageWork,
						   ipBlobContours := ipContourList,
						   stParams		  := BlobParameters,
						   hrPrev		  := hr);

hrWD := F_VN_StopWatchdog(hrWD, tRest => tRest, nFractionProcessed => nFraction);
END_METHOD

METHOD ReadParamUDINT : BOOL
VAR_INPUT
	Address : UDINT;
END_VAR

VAR_IN_OUT
	Value : UDINT;
	Valid : BOOL;
END_VAR
ReadParamUDINT := FALSE;
IF NOT _ReadData THEN
	_ReadData := TRUE;
ELSIF _ReadDataResult THEN
	_ReadData		:= FALSE;
	_ReadDataResult := FALSE;
	Valid			:= _ReadDataValid;
	Value			:= _ReadDataValue;
	ReadParamUDINT	:= TRUE;
END_IF
END_METHOD

METHOD SetParamUDINT : BOOL
VAR_INPUT
	Value	: UDINT;
	Address : UDINT;
END_VAR
SetParamUDINT := FALSE;
IF NOT _WriteData THEN
	_WriteData := TRUE;
	_WriteAddress := Address;
	_WriteValue := Value;
ELSIF _WriteDataDone THEN
	_WriteDataDone := FALSE;
	_WriteData := FALSE;
	SetParamUDINT := TRUE;
END_IF
END_METHOD

END_FUNCTION_BLOCK

// Vision/VisionTask/I_CameraBase
INTERFACE I_CameraBase

METHOD CyclicLogic
VAR_INPUT
END_VAR
END_METHOD

METHOD ProcessImage
VAR_INPUT
END_VAR
END_METHOD

END_INTERFACE

// Vision/VisionTask/FB_VisionCameraDetection
FUNCTION_BLOCK FB_VisionCameraDetection EXTENDS FB_VisionCameraBase
VAR

	// Iterator for Vision
	ipIterator : ITcVnForwardIterator;

	ipContourResultList : ITcVnContainer;
	ipContour			: ITcVnContainer;
	ipResultContainer	: ITcVnContainer;

	// Blob Detection
	///_BlobParams		 : TcVnParamsBlobDetection;
	Offset			 : TcVnPoint;


	//Configuration
	VisionTool : E_VisionTools;


	// Color
	nNewImageCounter : UINT;
	bTrigger		 : BOOL := TRUE;

	// Output
	Text		  : STRING(255);
	NumberOfBlobs : ULINT;
	BlobResults	  : ARRAY[1..100] OF ST_BlobResults;
	
	
END_VAR

METHOD ProcessImage
VAR
	ulint_ref		 : REFERENCE TO ULINT;
	i				 : ULINT;
	Rect			 : TcVnRectangle_UDINT;
	Text			 : STRING;
	Image_ID_NumText : STRING;
	nX				 : UDINT := 20;
	nY				 : UDINT := 50;
END_VAR
SUPER^.ProcessImage();

//Clear Results and set new results-Number of Blobs
MEMSET(ADR(BlobResults), 0, SIZEOF(BlobResults));
MEMSET(ADR(FeedbackResults), 0, SIZEOF(FeedbackResults));
ulint_ref REF= (NumberOfBlobs);
hr		  := F_VN_GetNumberOfElements(ipContainer := ipContourList, nNumberOfElements := ulint_ref, hrPrev := hr);
IF NumberOfBlobs > 0 THEN
	FOR i := 0 TO (NumberOfBlobs - 1) BY 1 DO
		hr := F_VN_GetAt_ITcVnContainer(ipSrcContainer	:= ipContourList,
										ipDestContainer := ipResultContainer,
										nIndex			:= i,
										hrPrev			:= hr);

		hr := F_VN_ContourArea(ipContour := ipResultContainer, fArea := BlobResults[i + 1].Area, hrPrev := hr);
		hr := F_VN_ContourCenterOfMass(ipContour := ipResultContainer, aCenterOfMass := BlobResults[i + 1].CenterOfMass, hrPrev := hr);

		//More items
		hr := F_VN_ContourCircularity(ipContour := ipResultContainer, fCircularity := BlobResults[i + 1].Circularity, hrPrev := hr);
		hr := F_VN_ContourConvexity(ipContour := ipResultContainer, fConvexity := BlobResults[i + 1].Convexity, hrPrev := hr);
		hr := F_VN_ContourEccentricity(ipContour := ipResultContainer, fEccentricity := BlobResults[i + 1].Eccentricity, hrPrev := hr);
		hr := F_VN_ContourInertiaRatio(ipContour := ipResultContainer, fInertiaRatio := BlobResults[i + 1].InertiaRatio, hrPrev := hr);
		hr := F_VN_ContourOrientation(ipContour := ipResultContainer, stOrientation := BlobResults[i + 1].Orientation, hrPrev := hr);
		hr := F_VN_ContourPerimeter(ipContour  := ipResultContainer,
									fPerimeter := BlobResults[i + 1].Perimeter,
									bClosed	   := TRUE,
									hrPrev	   := hr);

		hr := F_VN_ContourRoundness(ipContour := ipResultContainer, fRoundness := BlobResults[i + 1].Roundness, hrPrev := hr);

		//Copy the needed results into the return results
		FeedbackResults[i + 1].x		:= BlobResults[i + 1].CenterOfMass[0];
		FeedbackResults[i + 1].y		:= BlobResults[i + 1].CenterOfMass[1];
		FeedbackResults[i + 1].c		:= BlobResults[i + 1].Orientation.fAngle;
		FeedbackResults[i + 1].Distance := 0;
		FeedbackResults[i + 1].Pass		:= TRUE;
	END_FOR

	//Check the size of the buffer and the size to be copied
	IF SIZEOF(FeedbackResults) < SIZEOF(Results) THEN
		MEMCPY(ADR(Results), ADR(FeedbackResults), SIZEOF(FeedbackResults));
	ELSE
		MEMCPY(ADR(Results), ADR(FeedbackResults), SIZEOF(Results));
	END_IF
END_IF

//Return result number even if none found
NumberOfResults	 := TO_UDINT(NumberOfBlobs);
ResultsAvailable := TRUE;

(* Draw Result Image
// --------------------------------------------------------------*)
hr := F_VN_DrawContours(ipContourList,
						-1,
						ipImageRes,
						GVL_VisionColor.ColorGreen,
						3,
						hr);

IF NumberOfBlobs > 0 THEN
	FOR i := 0 TO (NumberOfBlobs - 1) DO
		hr := F_VN_GetAt_ITcVnContainer(ipSrcContainer	:= ipContourList,
										ipDestContainer := ipResultContainer,
										nIndex			:= i,
										hrPrev			:= hr);

		//hr	 := F_VN_UprightBoundingRectangle(ipResultContainer, Rect, hr);
		Text := TO_STRING(i + 1);
		hr	 := F_VN_PutText(Text,
							 ipImageRes,
							 TO_UDINT(BlobResults[i + 1].CenterOfMass[0]) - 20,
							 TO_UDINT(BlobResults[i + 1].CenterOfMass[1]) + 20,
							 TCVN_FT_HERSHEY_DUPLEX,
							 2,
							 GVL_VisionColor.ColorMagenta,
							 hr);
	END_FOR
END_IF

// Place the Block ID in White and in Black text in the upper left corner of the image
Image_ID_NumText := ULINT_TO_STRING(ImageCount);
hr				 := F_VN_PutTextExp(Image_ID_NumText,
									ipImageIn,
									nX,
									nY,
									TCVN_FT_HERSHEY_SIMPLEX,
									1.5,
									GVL_VisionColor.ColorWhite,
									3,
									TCVN_LT_8_CONNECTED,
									FALSE,
									hr);

hr := F_VN_PutTextExp(Image_ID_NumText,
					  ipImageIn,
					  nX,
					  nY + 50,
					  TCVN_FT_HERSHEY_SIMPLEX,
					  1.5,
					  GVL_VisionColor.ColorBlack,
					  3,
					  TCVN_LT_8_CONNECTED,
					  FALSE,
					  hr);

// Place the Block ID in White and in Black text in the upper left corner of the image
hr := F_VN_PutTextExp(Image_ID_NumText,
					  ipImageRes,
					  nX,
					  nY,
					  TCVN_FT_HERSHEY_SIMPLEX,
					  1.5,
					  GVL_VisionColor.ColorWhite,
					  3,
					  TCVN_LT_8_CONNECTED,
					  FALSE,
					  hr);

hr := F_VN_PutTextExp(Image_ID_NumText,
					  ipImageRes,
					  nX,
					  nY + 50,
					  TCVN_FT_HERSHEY_SIMPLEX,
					  1.5,
					  GVL_VisionColor.ColorBlack,
					  3,
					  TCVN_LT_8_CONNECTED,
					  FALSE,
					  hr);

// Display Input Image
hr := F_VN_TransformIntoDisplayableImage(ipImageIn, ipImageInDisp, hr);

// Display Result Image
hr := F_VN_TransformIntoDisplayableImage(ipImageRes, ipImageResDisp, hr);

// Display Threshold Image
hr := F_VN_TransformIntoDisplayableImage(ipImageWork, ipImageThresholdDisp, hr);
END_METHOD

METHOD PROTECTED Initialize : BOOL
VAR_INPUT
END_VAR
// Set Parameters

// --------------------------------------------------------------

// - Set fMaxArea to 100000 detect all circles or set it to 10000

// to detect only the small circles
BlobParameters.bFilterByArea		:= TRUE;
BlobParameters.fMinArea				:= 100;
BlobParameters.fMaxArea				:= 100000;
BlobParameters.bFilterByCircularity := TRUE;
BlobParameters.fMinCircularity		:= 0.80;
BlobParameters.fMinThreshold		:= 70;
BlobParameters.fThresholdStep		:= 0;

_LightBackground := TRUE;

Initialize := TRUE;
END_METHOD

END_FUNCTION_BLOCK

// Vision/VisionTask/FB_VisionCameraMonitor
FUNCTION_BLOCK FB_VisionCameraMonitor EXTENDS FB_VisionCameraBase
VAR
	// Video making properties
	_CameraID			  : UINT   := 1;
	_FramesPerSecond	  : UINT   := 10;
	_ImageSourceDirectory : STRING := 'C:\Images';
	_VideoOutputDirectory : STRING := 'C:\Videos';

	// Listener for JSON alarms with "Create
	VideoPlaybackControl :
		FB_VideoPlaybackControl := (ImageReductionFactor := 0.2, CameraID := _CameraID, ImageSourceDirectory := _ImageSourceDirectory,
									VideoOutputDirectory													 := _VideoOutputDirectory);
END_VAR

PROPERTY CameraID : UINT
SET
_CameraID := CameraID;
END_SET
END_PROPERTY

PROPERTY FramesPerSecond : UINT
SET
_FramesPerSecond := FramesPerSecond;
END_SET
END_PROPERTY

PROPERTY ImageSourceDirectory : STRING
SET
_ImageSourceDirectory := ImageSourceDirectory;
END_SET
END_PROPERTY

PROPERTY VideoOutputDirectory : STRING
SET
_VideoOutputDirectory := VideoOutputDirectory;
END_SET
END_PROPERTY

METHOD PUBLIC CyclicLogic
// Call the base here
SUPER^.CyclicLogic();

// Call the video playback here
VideoPlaybackControl.CyclicLogic();
END_METHOD

METHOD PROTECTED Initialize : BOOL
VAR_INPUT
END_VAR





Initialize := TRUE;
END_METHOD

METHOD PUBLIC  ProcessImage
hr := F_VN_GetPixelFormat(ipImageIn, PixelFormat, hr);
IF PixelFormat.nChannels = 3 THEN
	hr := F_VN_CopyImage(ipImageIn, ipImageRes, hr);
	hr := F_VN_ConvertColorSpace(ipImageRes,
								 ipImageIn,
								 TCVN_CST_RGB_TO_GRAY,
								 hr);
ELSE
	hr := F_VN_ConvertColorSpace(ipImageIn,
								 ipImageRes,
								 TCVN_CST_Gray_TO_RGB,
								 hr);
END_IF

// Display Input Image
hr := F_VN_CopyIntoDisplayableImage(ipImageIn, ipImageInDisp, hr);


VideoPlaybackControl.AddImage(ipImageIn := ipImageIn);
END_METHOD

END_FUNCTION_BLOCK
